// TIA Portal V20 export
TYPE "Interlock_Paletas_IKPAL_PLC"
   STRUCT
      BitDeVida : Bool;
      Libre_01 : Bool;
      Libre_02 : Bool;
      Libre_03 : Bool;
      Libre_04 : Bool;
      Libre_05 : Bool;
      Libre_06 : Bool;
      Libre_07 : Bool;
      IKPAL_Automatico : Bool;
      IKPAL_Manual : Bool;
      IKPAL_Error : Bool;
      Libre_13 : Bool;
      EntradaBultos_Automatico : Bool;
      SalidaPaletas_Automatico : Bool;
      Libre_16 : Bool;
      Libre_17 : Bool;
      Reserva_Array_18_B02 : Array[1..18] of Byte;
      NumeroPaletaSalida : UDInt;
      Reserva_Array_04_B24 : Array[1..4] of Byte;
      PermisoPreformado_PRV : Bool;
      FinPreformado_PRV : Bool;
      PermisoPreformado_PRV_Manual_Av : Bool;
      PermisoPreformado_PRV_Manual_Ret : Bool;
      Libre_284 : Bool;
      Libre_285 : Bool;
      Libre_286 : Bool;
      Libre_287 : Bool;
      AvisoPaleta_NXT : Bool;
      OrdenMarchaPaleta_NXT : Bool;
      AvisoPaleta_NXT_Manual_Av : Bool;
      AvisoPaleta_NXT_Manual_Ret : Bool;
      Libre_294 : Bool;
      Libre_295 : Bool;
      Libre_296 : Bool;
      Libre_297 : Bool;
      PeticionPaletaVacia : Bool;
      HorquillasExtendidas : Bool;
      HorquillasCentradas : Bool;
      PeticionAperturaPuertas : Bool;
      PuertasAccesoAbiertas : Bool;
      SubirMaqueta_Manual : Bool;
      BajarMaqueta_Manual : Bool;
      Libre_307 : Bool;
      Libre_310 : Bool;
      Libre_311 : Bool;
      Libre_312 : Bool;
      Libre_313 : Bool;
      Libre_314 : Bool;
      Libre_315 : Bool;
      Libre_316 : Bool;
      Libre_317 : Bool;
      Reserva_Array_06_B32 : Array[1..6] of Byte;
      MatriculaPaletaSalida : Array[1..10] of Byte;
      MckeyPaletaSalida : Array[1..8] of Byte;
   END_STRUCT;
END_TYPE
